Yaskawa INFORM job: R1_W53-A2(90,90).JBI

/JOB
//NAME R1_W53-A2(90,90)
///FOLDERNAME KRIS-SCIANA
//POS
///NPOS 54,54,0,2,0,0
///TOOL 0
///POSTYPE PULSE
///PULSE
C00000=-114985,85289,38053,-11,81830,11658
C00001=-121260,37195,8937,-6676,74802,26688
C00002=-121230,45828,34626,-7184,63509,27357
C00003=-122241,52002,44250,-6962,60690,27149
C00004=-122994,54347,48026,-6736,59521,26928
C00005=-122980,56191,50093,-6764,59200,26953
C00006=-122635,54705,48425,-6883,59484,27070
C00007=-115735,72932,70832,-23348,64424,33496
C00008=-116402,72721,70578,-23183,64281,33259
C00009=-115735,72932,70832,-23348,64424,33496
C00010=-122958,68544,61895,-6055,65181,26969
C00011=-122958,69252,63866,-6096,64336,27014
C00012=-122949,69675,63073,-6066,65039,26981
C00013=-122579,66793,58372,-6109,66471,27043
C00014=-121633,60489,47853,-6244,69759,27215
C00015=-120725,83956,80574,6404,98515,-580
C00016=-120725,89416,91854,6335,94404,-790
C00017=-120713,89375,93303,6323,93490,-831
C00018=-120720,87086,89636,6338,94570,-781
C00019=-120722,95358,100430,6313,92192,-901
C00020=-120734,88731,92151,6326,93874,-820
C00021=-120725,89405,91869,6335,94389,-791
C00022=-120725,83940,80582,6404,98503,-580
C00023=-121680,62807,51682,4317,62008,41600
C00024=-120821,65218,58094,4083,59262,41827
C00025=-120969,55622,51477,4463,52952,41513
C00026=-120602,66928,60297,4016,58777,41895
C00027=-120553,64941,58336,3989,58959,41921
C00028=-121930,55328,51051,4944,53118,41119
C00029=-120433,63699,54964,4849,63853,36385
C00030=-120724,64354,52136,4865,65942,36365
C00031=-120500,45873,5560,4425,85036,37161
C00032=-145452,78104,42568,11880,81321,28736
C00033=-156803,-4457,-23706,38570,72296,36252
C00034=-145388,-53797,-49151,49039,52473,43059
C00035=-153251,-10941,-15086,57455,90636,31659
C00036=-152418,-13006,-14739,57396,89421,31325
C00037=-155236,18881,12248,62852,109135,25204
C00038=-153863,23836,20908,62091,106910,24239
C00039=-146924,19108,24533,59569,99597,23263
C00040=-144263,17292,25920,58605,96794,22892
C00041=-141947,-1894,10843,60671,86000,25676
C00042=-139417,-1625,8723,55159,86485,19479
C00043=-141210,-1964,11178,60745,85417,25706
C00044=-141032,-725,11836,60750,85424,25829
C00045=-140129,-1341,12357,60163,85946,18209
C00046=-141965,-2741,12214,62321,84861,23993
C00047=-144263,17292,25920,58605,96794,22892
C00048=-147702,18037,20518,58716,100901,23729
C00049=-152047,-14155,-11854,60653,87045,29536
C00050=-145388,-53797,-49151,49039,52473,43059
C00051=-145388,-55037,-56302,47016,55043,44620
C00052=-145388,-100918,-92455,47016,55043,44620
C00053=-19781,-100918,-92455,47016,55043,44620
BC00000=80451,971848,1068220
BC00001=75633,679574,1068222
BC00002=75633,679574,1068222
BC00003=75633,679574,1068222
BC00004=75633,679574,1068218
BC00005=75633,679574,1068218
BC00006=75633,679574,1068222
BC00007=75633,679574,1068222
BC00008=75633,679574,1068222
BC00009=75633,679574,1068222
BC00010=75633,679574,1068222
BC00011=75633,679574,1068222
BC00012=75633,679574,1068222
BC00013=75633,679574,1068222
BC00014=75633,679574,1068222
BC00015=38930,720293,1068222
BC00016=39846,720947,1068222
BC00017=40088,721099,1068221
BC00018=40213,721209,1068222
BC00019=40213,721209,1068222
BC00020=47744,721219,1068222
BC00021=47378,720957,1068222
BC00022=46461,720303,1068222
BC00023=56547,671045,1068222
BC00024=54020,674200,1068222
BC00025=53009,675462,1068222
BC00026=53009,675462,1068222
BC00027=53009,675462,1068222
BC00028=53009,675462,1068222
BC00029=48193,678393,1068222
BC00030=50572,675072,1068222
BC00031=50572,675072,1068222
BC00032=50572,675072,1068222
BC00033=18769,740965,1068222
BC00034=876,778038,1068222
BC00035=876,778038,1068222
BC00036=876,778038,1068222
BC00037=876,778038,1068222
BC00038=876,778038,1068222
BC00039=876,778038,1068222
BC00040=876,778038,1068222
BC00041=876,777537,1068222
BC00042=876,777857,1068219
BC00043=876,778479,1068222
BC00044=876,778479,1068222
BC00045=876,777857,1068219
BC00046=876,777857,1068219
BC00047=876,778038,1068222
BC00048=876,778038,1068222
BC00049=876,778038,1068222
BC00050=876,778038,1068222
BC00051=876,778038,1068222
BC00052=876,778038,1068222
BC00053=876,700798,1068222
///POSTYPE BASE
///RECTAN
///RCONF 0,0,0,0,0,0,0,0,0,0,0,0,0,0,0,0,0,0,0,0,0,0,0,0
P00006=0.222,-3.123,-1.508,0.0000,0.0000,0.0000
P00022=0.222,-3.123,-1.508,0.0000,0.0000,0.0000
//INST
///DATE 2024/07/24 16:32
///ATTR SC,RW
///GROUP1 RB1,BS1
NOP
'Path S980
SFTOF
MOVJ C00000 BC00000 VJ=100.00
MOVJ C00001 BC00001 VJ=100.00
MOVJ C00002 BC00002 VJ=20.00
MOVL C00003 BC00003 V=100.0
MOVL C00004 BC00004 V=60.0
REFP 3 C00005 BC00005
CALL JOB:SEARCH-R1
SET P022 P006
SFTON P022
MOVL C00006 BC00006 V=60.0
MOVL C00007 BC00007 V=60.0
REFP 3 C00008 BC00008
CALL JOB:SEARCH-R1
SET P022 P006
SFTON P022
MOVL C00009 BC00009 V=60.0
MOVL C00010 BC00010 V=60.0
REFP 3 C00011 BC00011
CALL JOB:SEARCH-R1
SET P022 P006
SFTON P022
MOVL C00012 BC00012 V=60.0
MOVL C00013 BC00013 V=100.0
MOVL C00014 BC00014 V=100.0
'Path W981
SFTOF
SFTON P022
MOVL C00015 BC00015 V=100.0
MOVL C00016 BC00016 V=100.0
MOVL C00017 BC00017 V=100.0 PL=0
REFP 1 C00018 BC00018
REFP 2 C00019 BC00019
MACRO1 MJ#(0) ARGF7
ARCON
MOVL C00020 BC00020 V=10.0
ARCOF
MOVL C00021 BC00021 V=100.0
MOVL C00022 BC00022 V=250.0
SFTOF
'Path W982
SFTOF
SFTON P022
MOVJ C00023 BC00023 VJ=20.00
MOVL C00024 BC00024 V=133.3
MOVL C00025 BC00025 V=100.0 PL=0
REFP 1 C00026 BC00026
REFP 2 C00027 BC00027
MACRO1 MJ#(0) ARGF7
ARCON
MOVL C00028 BC00028 V=8.3
ARCOF
MOVL C00029 BC00029 V=166.7
MOVL C00030 BC00030 V=250.0
SFTOF
'Path VIA1071
SFTOF
MOVJ C00031 BC00031 VJ=20.00
'Path VIA1072
SFTOF
MOVJ C00032 BC00032 VJ=20.00
MOVJ C00033 BC00033 VJ=20.00
MOVJ C00034 BC00034 VJ=20.00
SFTOF
MOVJ C00035 BC00035 VJ=10.00
MOVJ C00036 BC00036 VJ=20.00
MOVJ C00037 BC00037 VJ=10.00
MOVJ C00038 BC00038 VJ=15.00
'Path VIA1069
SFTOF
'Path VIA1067
SFTOF
MOVJ C00039 BC00039 VJ=15.00
MOVJ C00040 BC00040 VJ=10.00
'Path W983
SFTOF
SFTON P022
MOVL C00041 BC00041 V=100.0
MOVL C00042 BC00042 V=100.0 PL=0
REFP 1 C00043 BC00043
REFP 2 C00044 BC00044
MACRO1 MJ#(0) ARGF7
ARCON
MOVL C00045 BC00045 V=10.0
ARCOF
MOVL C00046 BC00046 V=100.0
SFTOF
'Path VIA1063
SFTOF
MOVJ C00047 BC00047 VJ=10.00
'Path VIA1064
SFTOF
MOVJ C00048 BC00048 VJ=10.00
'Path VIA1065
SFTOF
MOVJ C00049 BC00049 VJ=10.00
'Path VIA1066
SFTOF
MOVJ C00050 BC00050 VJ=20.00
MOVJ C00051 BC00051 VJ=100.00
'COMMENT
MOVJ C00052 BC00052 VJ=100.00
MOVJ C00053 BC00053 VJ=100.00
END
